// TIA Portal V15.1 export
// export: Created 2020-06-12T07:35:49.4599609Z, ExportSetting None, DisplayName Totally Integrated Automation Portal, DisplayVersion V15.1, DisplayName TIA Portal Openness, DisplayVersion V15.1, DisplayName STEP 7 Professional, DisplayVersion V15.1, DisplayName STEP 7 Safety, DisplayVersion V15.1, DisplayName WinCC Advanced, DisplayVersion V15.1
FUNCTION "ContrFast_call" : Void   // FC177, FBD
TITLE = Fast PID/SMC controllers
{ S7_Optimized_Access := 'TRUE' }
// stored: SetENOAutomatically False
BEGIN

REGION Network 1: Main line pressure control: PID controller
   // ES1LC1.M02 - .M03
   // ES1LC1.PT01
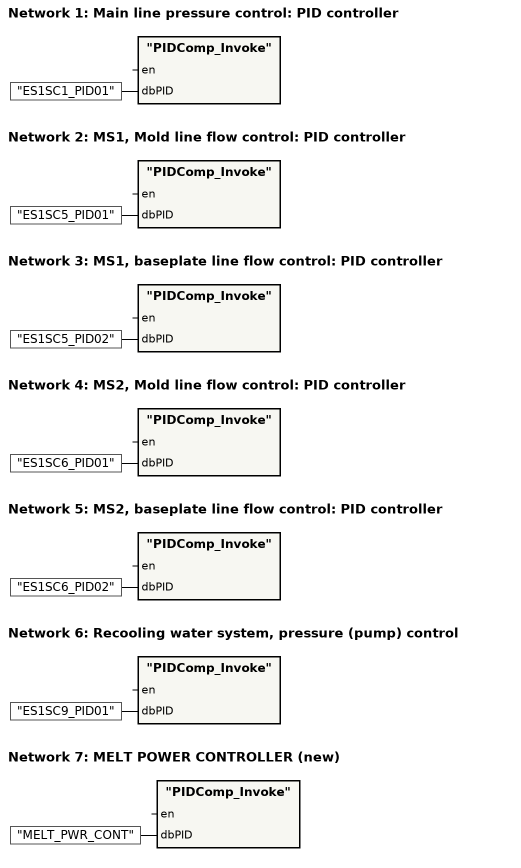
   "PIDComp_Invoke"(dbPID := "ES1SC1_PID01");
END_REGION

REGION Network 2: MS1, Mold line flow control: PID controller
   // ES1LC5.CV01
   // ES1LC5.FT01
   "PIDComp_Invoke"(dbPID := "ES1SC5_PID01");
END_REGION

REGION Network 3: MS1, baseplate line flow control: PID controller
   // ES1LC5.CV02
   // ES1LC5.FT02
   "PIDComp_Invoke"(dbPID := "ES1SC5_PID02");
END_REGION

REGION Network 4: MS2, Mold line flow control: PID controller
   // ES1LC5.CV01
   // ES1LC5.FT01
   "PIDComp_Invoke"(dbPID := "ES1SC6_PID01");
END_REGION

REGION Network 5: MS2, baseplate line flow control: PID controller
   // ES1LC6.CV02
   // ES1LC6.FT02
   "PIDComp_Invoke"(dbPID := "ES1SC6_PID02");
END_REGION

REGION Network 6: Recooling water system, pressure (pump) control
   "PIDComp_Invoke"(dbPID := "ES1SC9_PID01");
END_REGION

REGION Network 7: MELT POWER CONTROLLER (new)
   "PIDComp_Invoke"(dbPID := "MELT_PWR_CONT");
END_REGION
END_FUNCTION
